// TwinCAT 3 PLC project PLC
// ProgramVersion: 3.1.4024.0
// libraries:
//   Tc2_MC2, * (Beckhoff Automation GmbH)
//   Tc2_Standard, * (Beckhoff Automation GmbH)
//   Tc2_System, * (Beckhoff Automation GmbH)
//   Tc2_Utilities, * (Beckhoff Automation GmbH)
//   Tc3_EventLogger, * (Beckhoff Automation GmbH)
//   Tc3_Module, * (Beckhoff Automation GmbH)
//   Util, * (System)
// project tree:
//   DUTs/ E_State.TcDUT, ST_CarrierSetpoint.TcDUT, ST_LEDButton.TcDUT, ST_MachineModuleInputs.TcDUT
//   / PlcTask.TcTTO (not stored)
//   POUs/ FB_CarrierStop.TcPOU, FB_CarrierReset.TcPOU, FB_CarrierAbsMove.TcPOU, FB_Machine.TcPOU, FB_Alarm.TcPOU, F_E_State_To_String.TcPOU, MAIN.TcPOU, PRG_LoadTwinSAFE.TcPOU
// real-time tasks:
//   TASK PlcTask: cycle T#10ms, priority 20, ADS port 350
// motion (NC):
//   TASK NC-Task 1 SAF: cycle T#2ms, priority 4, ADS port 501
//   TASK NC-Task 1 SVB: cycle T#10ms, priority 8, ADS port 511
//   AXIS X (id 1)
//     Dynamic: AccelerationMaximum=100000, DecelerationMaximum=100000, Acceleration=3082.5, Deceleration=3082.5, Jerk=9247.5
//     Velo: RefSearch=20.55, RefSync=20.55, SlowManual=102.75, FastManual=616.5, Fast=2055, Maximum=2055
//     OtherSettings: AllowMotionCmdToSlave=true
//     encoder EncType=19
//       EncPara: ScaleFactorNumerator=100, ScaleFactorDenominator=1048576, MaxCount=#xffffffff
//         SoftEndMinControl: Enable=true
//         SoftEndMaxControl: Enable=true, Range=2000
//     encoder EncId=129, EncType=5
//       EncPara: ScaleFactorNumerator=10, ScaleFactorDenominator=4096, Offset=-1035.7471, MaxCount=#xffffffff, ReferenceSystem=1
//         Inc: RefSoftSyncMask=#x0000ffff
//     drive DrvType=16
//       DrvPara: MaxCount=#xffffffff, DriveControlDWord=#x00020100
//         Analog: VeloReferenz=2260.5, VeloScale=32, TorqueSetpointScale=10, ScaleFactorActTorque=0.1
//         TimeComp: TaskDelayCycles=1
//     controller CtrType=1
//       CtrPara: PriorControlFactor=1
//         Observer: BandWidth=20
//   AXIS Z (id 2)
//     Dynamic: AccelerationMaximum=100000, DecelerationMaximum=100000, Acceleration=3082.5, Deceleration=3082.5, Jerk=9247.5
//     Velo: RefSearch=20.55, RefSync=20.55, SlowManual=102.75, FastManual=616.5, Fast=2055, Maximum=2055
//     OtherSettings: AllowMotionCmdToSlave=true
//     encoder EncType=19
//       EncPara: ScaleFactorNumerator=100, ScaleFactorDenominator=1048576, MaxCount=#xffffffff
//         SoftEndMinControl: Enable=true
//         SoftEndMaxControl: Enable=true, Range=1500
//     drive DrvType=16
//       DrvPara: MaxCount=#xffffffff, DriveControlDWord=#x00020100
//         Analog: VeloReferenz=2260.5, VeloScale=32, TorqueSetpointScale=10, ScaleFactorActTorque=0.1
//         TimeComp: TaskDelayCycles=1
//     controller CtrType=1
//       CtrPara: PriorControlFactor=1
//         Observer: BandWidth=20
// I/O:
//   DEVICE Real IO, AmsNetId 0.0.0.0.2.1
//     Term 1 (EK1200) [EK1200-5000 EtherCAT Power supply (2A E-Bus)]
//       Machine Safety Controller (EL6910) [EL6910, TwinSAFE PLC]
//       Operator Panel Safe In (EL1904) [EL1904, 4 Ch. Safety Input 24V, TwinSAFE]
//         modules: Module 1 (FSOES)
//   DEVICE Sim IO, AmsNetId 0.0.0.0.3.1
//     Machine A (EK1100) [EK1100 EtherCAT Coupler (2A E-Bus)]
//       Machine A Safe In (EL1904) [EL1904, 4 Ch. Safety Input 24V, TwinSAFE]
//         modules: Module 1 (FSOES)
//       Machine A Safe out (EL2904) [EL2904, 4 Ch. Safety Output 24V, 0.5A, TwinSAFE]
//         modules: Module 1 (FSOES), Module 2 (DO)
//       Robot (EL2002) [EL2002 2Ch. Dig. Output 24V, 0.5A]
//       Part Status (EL1002) [EL1002 2Ch. Dig. Input 24V, 3ms]
//     Machine B (EK1100) [EK1100 EtherCAT Coupler (2A E-Bus)]
//       Machine B Safe In (EL1904) [EL1904, 4 Ch. Safety Input 24V, TwinSAFE]
//         modules: Module 1 (FSOES)
//       Machine B Safe out (EL2904) [EL2904, 4 Ch. Safety Output 24V, 0.5A, TwinSAFE]
//         modules: Module 1 (FSOES), Module 2 (DO)
//       QC Check (EL3001) [EL3001 1Ch. Ana. Input +/-10V]
//     Machine C (EK1100) [EK1100 EtherCAT Coupler (2A E-Bus)]
//       Machine C Safe In (EL1904) [EL1904, 4 Ch. Safety Input 24V, TwinSAFE]
//         modules: Module 1 (FSOES)
//       Machine C Safe out (EL2904) [EL2904, 4 Ch. Safety Output 24V, 0.5A, TwinSAFE]
//         modules: Module 1 (FSOES), Module 2 (DO)
//       Bending (EL4001) [EL4001 1Ch. Ana. Output 0-10V, 12bit]
//     Machine D (EK1100) [EK1100 EtherCAT Coupler (2A E-Bus)]
//       Machine D Safe In (EL1904) [EL1904, 4 Ch. Safety Input 24V, TwinSAFE]
//         modules: Module 1 (FSOES)
//       Machine D Safe out (EL2904) [EL2904, 4 Ch. Safety Output 24V, 0.5A, TwinSAFE]
//         modules: Module 1 (FSOES), Module 2 (DO)
//       Carrier X Safety Encoder (EL5001-0090) [EL5001-0090 1Ch. SSI Encoder, TwinSAFE SC]
//         modules: Module 1 (EL5001-0090)
//       Carrier X Axis (EL7211-9014) [EL7211-9014 1Ch. MDP742 Servo motor output stage with OCT (50V, 4.5A RMS) and STO input]
//       Carrier Z Axis (EL7211-9014) [EL7211-9014 1Ch. MDP742 Servo motor output stage with OCT (50V, 4.5A RMS) and STO input]
//       Carrier Gripper (EL2002) [EL2002 2Ch. Dig. Output 24V, 0.5A]
//   DEVICE CP Buttons
// variable links:
//   Real IO <-> Sim IO/Machine A (EK1100)/Machine A Safe In (EL1904)
//     Term 1 (EK1200)/Machine Safety Controller (EL6910)/ConnectionInputs/TwinSafeGroup1.Machine A Safe In (EL1904) - Module 1 (FSOES)_32 TxPDO <-> Module 1 (FSOES)/RxPDO/FSOE
//     Term 1 (EK1200)/Machine Safety Controller (EL6910)/ConnectionOutputs/TwinSafeGroup1.Machine A Safe In (EL1904) - Module 1 (FSOES)_32 RxPDO <-> Module 1 (FSOES)/TxPDO/FSOE
//   Real IO <-> Sim IO/Machine B (EK1100)/Machine B Safe In (EL1904)
//     Term 1 (EK1200)/Machine Safety Controller (EL6910)/ConnectionOutputs/TwinSafeGroup1.Machine B Safe In (EL1904) - Module 1 (FSOES)_34 RxPDO <-> Module 1 (FSOES)/TxPDO/FSOE
//   Real IO <-> Sim IO/Machine B (EK1100)/Machine B Safe out (EL2904)
//     Term 1 (EK1200)/Machine Safety Controller (EL6910)/ConnectionInputs/TwinSafeGroup1.Machine B Safe out (EL2904) - Module 1 (FSOES)_35 TxPDO <-> Module 1 (FSOES)/RxPDO/FSOE
//   Real IO <-> Sim IO/Machine C (EK1100)/Machine C Safe In (EL1904)
//     Term 1 (EK1200)/Machine Safety Controller (EL6910)/ConnectionInputs/TwinSafeGroup1.Machine C Safe In (EL1904) - Module 1 (FSOES)_36 TxPDO <-> Module 1 (FSOES)/RxPDO/FSOE
//     Term 1 (EK1200)/Machine Safety Controller (EL6910)/ConnectionOutputs/TwinSafeGroup1.Machine C Safe In (EL1904) - Module 1 (FSOES)_36 RxPDO <-> Module 1 (FSOES)/TxPDO/FSOE
//   Real IO <-> Sim IO/Machine C (EK1100)/Machine C Safe out (EL2904)
//     Term 1 (EK1200)/Machine Safety Controller (EL6910)/ConnectionInputs/TwinSafeGroup1.Machine C Safe out (EL2904) - Module 1 (FSOES)_37 TxPDO <-> Module 1 (FSOES)/RxPDO/FSOE
//     Term 1 (EK1200)/Machine Safety Controller (EL6910)/ConnectionOutputs/TwinSafeGroup1.Machine C Safe out (EL2904) - Module 1 (FSOES)_37 RxPDO <-> Module 1 (FSOES)/TxPDO/FSOE
//   Real IO <-> Sim IO/Machine D (EK1100)/Carrier X Safety Encoder (EL5001-0090)
//     Term 1 (EK1200)/Machine Safety Controller (EL6910)/ConnectionInputs/TwinSafeGroup1.Carrier X Safety Encoder (EL5001-0090) - Module 1 (EL5001-0090)_48 TxPDO <-> Module 1 (EL5001-0090)/TSC Master Message/TSC
//     Term 1 (EK1200)/Machine Safety Controller (EL6910)/ConnectionOutputs/TwinSafeGroup1.Carrier X Safety Encoder (EL5001-0090) - Module 1 (EL5001-0090)_48 RxPDO <-> Module 1 (EL5001-0090)/TSC Slave Message/TSC
//   Sim IO <-> Real IO/Term 1 (EK1200)/Machine Safety Controller (EL6910)
//     Machine A (EK1100)/Machine A Safe out (EL2904)/Module 1 (FSOES)/RxPDO/FSOE <-> ConnectionInputs/TwinSafeGroup1.Machine A Safe out (EL2904) - Module 1 (FSOES)_33 TxPDO
//     Machine A (EK1100)/Machine A Safe out (EL2904)/Module 1 (FSOES)/TxPDO/FSOE <-> ConnectionOutputs/TwinSafeGroup1.Machine A Safe out (EL2904) - Module 1 (FSOES)_33 RxPDO
//     Machine B (EK1100)/Machine B Safe In (EL1904)/Module 1 (FSOES)/RxPDO/FSOE <-> ConnectionInputs/TwinSafeGroup1.Machine B Safe In (EL1904) - Module 1 (FSOES)_34 TxPDO
//     Machine B (EK1100)/Machine B Safe out (EL2904)/Module 1 (FSOES)/TxPDO/FSOE <-> ConnectionOutputs/TwinSafeGroup1.Machine B Safe out (EL2904) - Module 1 (FSOES)_35 RxPDO
//     Machine D (EK1100)/Machine D Safe In (EL1904)/Module 1 (FSOES)/RxPDO/FSOE <-> ConnectionInputs/TwinSafeGroup1.Machine D Safe In (EL1904) - Module 1 (FSOES)_38 TxPDO
//     Machine D (EK1100)/Machine D Safe In (EL1904)/Module 1 (FSOES)/TxPDO/FSOE <-> ConnectionOutputs/TwinSafeGroup1.Machine D Safe In (EL1904) - Module 1 (FSOES)_38 RxPDO
//     Machine D (EK1100)/Machine D Safe out (EL2904)/Module 1 (FSOES)/RxPDO/FSOE <-> ConnectionInputs/TwinSafeGroup1.Machine D Safe out (EL2904) - Module 1 (FSOES)_39 TxPDO
//     Machine D (EK1100)/Machine D Safe out (EL2904)/Module 1 (FSOES)/TxPDO/FSOE <-> ConnectionOutputs/TwinSafeGroup1.Machine D Safe out (EL2904) - Module 1 (FSOES)_39 RxPDO
//   (this object) <-> Sim IO/Machine D (EK1100)/Carrier X Axis (EL7211-9014)
//     Drive/Inputs/In/nDataIn1 <-> DRV Following error actual value/Following error actual value
//     Drive/Inputs/In/nDataIn3[0] <-> DRV Torque actual value/Torque actual value
//     Drive/Inputs/In/nDcOutputTime <-> InfoData/DcOutputShift
//     Drive/Inputs/In/nState1 <-> DRV Statusword/Statusword
//     Drive/Inputs/In/nState2 <-> DRV Statusword/Statusword @bit 8
//     Drive/Inputs/In/nState4 @bit 1 <-> WcState/InputToggle
//     Drive/Inputs/In/nState4 <-> WcState/WcState
//     Drive/Outputs/Out/nCtrl1 <-> DRV Controlword/Controlword
//     Drive/Outputs/Out/nCtrl2 <-> DRV Controlword/Controlword @bit 8
//     Drive/Outputs/Out/nDataOut1 <-> DRV Target position/Target position
//     EL7211/Inputs/In/nDataIn1 <-> FB Position/Position
//     EL7211/Inputs/In/nDcInputTime <-> InfoData/DcInputShift
//     EL7211/Inputs/In/nState4 @bit 1 <-> WcState/InputToggle
//     EL7211/Inputs/In/nState4 <-> WcState/WcState
//   (this object) <-> Sim IO/Machine D (EK1100)/Carrier X Safety Encoder (EL5001-0090)
//     EL5001-0090/Inputs/In/nDataIn1 <-> SSI Inputs/Counter value
//     EL5001-0090/Inputs/In/nState1 <-> SSI Inputs/Status/Data error
//     EL5001-0090/Inputs/In/nState1 @bit 1 <-> SSI Inputs/Status/Frame error
//     EL5001-0090/Inputs/In/nState1 @bit 2 <-> SSI Inputs/Status/Power failure
//     EL5001-0090/Inputs/In/nState2 @bit 5 <-> SSI Inputs/Status/Sync error
//     EL5001-0090/Inputs/In/nState2 @bit 6 <-> SSI Inputs/Status/TxPDO State
//     EL5001-0090/Inputs/In/nState2 @bit 7 <-> SSI Inputs/Status/TxPDO Toggle
//     EL5001-0090/Inputs/In/nState4 @bit 1 <-> WcState/InputToggle
//     EL5001-0090/Inputs/In/nState4 <-> WcState/WcState
//   (this object) <-> Sim IO/Machine D (EK1100)/Carrier Z Axis (EL7211-9014)
//     Drive/Inputs/In/nDataIn1 <-> DRV Following error actual value/Following error actual value
//     Drive/Inputs/In/nDataIn3[0] <-> DRV Torque actual value/Torque actual value
//     Drive/Inputs/In/nDcOutputTime <-> InfoData/DcOutputShift
//     Drive/Inputs/In/nState1 <-> DRV Statusword/Statusword
//     Drive/Inputs/In/nState2 <-> DRV Statusword/Statusword @bit 8
//     Drive/Inputs/In/nState4 @bit 1 <-> WcState/InputToggle
//     Drive/Inputs/In/nState4 <-> WcState/WcState
//     Drive/Outputs/Out/nCtrl1 <-> DRV Controlword/Controlword
//     Drive/Outputs/Out/nCtrl2 <-> DRV Controlword/Controlword @bit 8
//     Drive/Outputs/Out/nDataOut1 <-> DRV Target position/Target position
//     EL7211/Inputs/In/nDataIn1 <-> FB Position/Position
//     EL7211/Inputs/In/nDcInputTime <-> InfoData/DcInputShift
//     EL7211/Inputs/In/nState4 @bit 1 <-> WcState/InputToggle
//     EL7211/Inputs/In/nState4 <-> WcState/WcState
//   (this object) <-> Real IO
//     Term 1 (EK1200)/Machine Safety Controller (EL6910)/ConnectionInputs/TwinSafeGroup1.Operator Panel Safe In (EL1904) - Module 1 (FSOES)_43 TxPDO <-> Term 1 (EK1200)/Operator Panel Safe In (EL1904)/Module 1 (FSOES)/RxPDO/FSOE
//     Term 1 (EK1200)/Machine Safety Controller (EL6910)/ConnectionOutputs/TwinSafeGroup1.Operator Panel Safe In (EL1904) - Module 1 (FSOES)_43 RxPDO <-> Term 1 (EK1200)/Operator Panel Safe In (EL1904)/Module 1 (FSOES)/TxPDO/FSOE
//     Term 1 (EK1200)/Operator Panel Safe In (EL1904)/Module 1 (FSOES)/RxPDO/FSOE <-> Term 1 (EK1200)/Machine Safety Controller (EL6910)/ConnectionInputs/TwinSafeGroup1.Operator Panel Safe In (EL1904) - Module 1 (FSOES)_43 TxPDO
//     Term 1 (EK1200)/Operator Panel Safe In (EL1904)/Module 1 (FSOES)/TxPDO/FSOE <-> Term 1 (EK1200)/Machine Safety Controller (EL6910)/ConnectionOutputs/TwinSafeGroup1.Operator Panel Safe In (EL1904) - Module 1 (FSOES)_43 RxPDO
//   PLC Instance <-> CP Buttons/Box 0 (CPX8XX)
//     PlcTask Inputs/MAIN.Machine.LocalEstop <-> Term 1 (CPx9xx-4)/Channel 1/Estop
//     PlcTask Inputs/MAIN.Machine.Reset.Button <-> Term 1 (CPx9xx-4)/Channel 1/BlueBtn
//     PlcTask Inputs/MAIN.Machine.Start.Button <-> Term 1 (CPx9xx-4)/Channel 1/GreenBtn
//     PlcTask Inputs/MAIN.Machine.Stop.Button <-> Term 1 (CPx9xx-4)/Channel 1/RedBtn
//     PlcTask Outputs/MAIN.Machine.Reset.LED <-> Term 1 (CPx9xx-4)/Channel 1/BlueBtnLight
//     PlcTask Outputs/MAIN.Machine.Start.LED <-> Term 1 (CPx9xx-4)/Channel 1/GreenBtnLight
//     PlcTask Outputs/MAIN.Machine.Stop.LED <-> Term 1 (CPx9xx-4)/Channel 1/RedBtnLight
//   PLC Instance <-> Real IO/Term 1 (EK1200)/Machine Safety Controller (EL6910)
//     PlcTask Inputs/MAIN.Machine.TwinSAFEGroupState <-> TwinSAFE Group Info Data/TwinSafeGroup1 Info Data/State
//     PlcTask Inputs/MAIN.Machine.TwinSAFE_Machine_A_Estop_State <-> Function Block Info Data/TwinSafeGroup1.MachineA.Machine_A.FBEstop1 Info Data/State
//     PlcTask Inputs/MAIN.Machine.TwinSAFE_Machine_B_Estop_State <-> Function Block Info Data/TwinSafeGroup1.MachineB.Machine_B.FBEstop1 Info Data/State
//     PlcTask Inputs/MAIN.Machine.TwinSAFE_Machine_C_Estop_State <-> Function Block Info Data/TwinSafeGroup1.MachineC.Machine_C.FBEstop1 Info Data/State
//     PlcTask Inputs/MAIN.Machine.TwinSAFE_Machine_D_Estop_State <-> Function Block Info Data/TwinSafeGroup1.MachineD.Machine_D_Estop Info Data/State
//     PlcTask Inputs/PRG_LoadTwinSAFE.ProjectCRC <-> Device Info Data/Project CRC
//     PlcTask Inputs/PRG_LoadTwinSAFE.WcState <-> WcState/WcState
//     PlcTask Outputs/MAIN.Machine.TwinSAFEGroupErrAck <-> StandardOutputs/TwinSafeGroup1.ErrorAcknowledgement_1
//     PlcTask Outputs/MAIN.Machine.TwinSAFEGroupRun <-> StandardOutputs/TwinSafeGroup1.Run_2
//     PlcTask Outputs/MAIN.Machine.TwinSAFE_ResetAllEstopZones <-> StandardOutputs/TwinSafeGroup1.ResetAllZones_55
//     PlcTask Outputs/MAIN.Machine.TwinSAFE_X_Axis_ActPos <-> StandardOutputs/TwinSafeGroup1.X_ActPosFromPLC_51
//   PLC Instance <-> Sim IO/Machine A (EK1100)/Machine A Safe In (EL1904)
//     PlcTask Inputs/MAIN.Machine.MachineAIn.EstopBtn <-> Module 1 (FSOES)/TxPDO/FSOE/E-Stop PB
//     PlcTask Inputs/MAIN.Machine.MachineAIn.LightCurtain <-> Module 1 (FSOES)/TxPDO/FSOE/Light Curtain
//   PLC Instance <-> Sim IO/Machine B (EK1100)/Machine B Safe In (EL1904)
//     PlcTask Inputs/MAIN.Machine.MachineBIn.EstopBtn <-> Module 1 (FSOES)/TxPDO/FSOE/E-Stop PB
//     PlcTask Inputs/MAIN.Machine.MachineBIn.LightCurtain <-> Module 1 (FSOES)/TxPDO/FSOE/Light Curtain
//   PLC Instance <-> Sim IO/Machine C (EK1100)/Machine C Safe In (EL1904)
//     PlcTask Inputs/MAIN.Machine.MachineCIn.EstopBtn <-> Module 1 (FSOES)/TxPDO/FSOE/E-Stop PB
//     PlcTask Inputs/MAIN.Machine.MachineCIn.LightCurtain <-> Module 1 (FSOES)/TxPDO/FSOE/Light Curtain
//   PLC Instance <-> Sim IO/Machine D (EK1100)/Carrier Gripper (EL2002)
//     PlcTask Outputs/MAIN.Machine.Machine_D_Carrier_Gripper <-> Fingers/Output
//   PLC Instance <-> Sim IO/Machine D (EK1100)/Machine D Safe In (EL1904)
//     PlcTask Inputs/MAIN.Machine.MachineDIn.EstopBtn <-> Module 1 (FSOES)/TxPDO/FSOE/E-Stop PB
//   PLC Instance <-> NC-Task 1 SAF/Axes/X
//     PlcTask Inputs/MAIN.Machine.X_Axis.NcToPlc <-> Outputs/ToPlc
//     PlcTask Outputs/MAIN.Machine.X_Axis.PlcToNc <-> Inputs/FromPlc
//   PLC Instance <-> NC-Task 1 SAF/Axes/Z
//     PlcTask Inputs/MAIN.Machine.Z_Axis.NcToPlc <-> Outputs/ToPlc
//     PlcTask Outputs/MAIN.Machine.Z_Axis.PlcToNc <-> Inputs/FromPlc

// ---- DUTs/E_State.TcDUT
{attribute 'qualified_only'}
{attribute 'strict'}
TYPE
	E_State :
	(
		Init := 0,
		Idel,
		Enable,
		MoveToHome,			// Move X and Z to home poisition
		WaitForAToBeReady,	// Wait at home postion for A to be ready
		MoveToAPickPos,		// Move X and Z to A position
		PickFromA,			// Close Grippers
		MoveToBWaitPos,		// Move X and Z to safe B position
		WaitForBToBeReady,
		MoveToBPlacePosition,	// Move X and Z to B Position
		PlaceOnB,				// Open grippers
		MoveToBWorkPos,			// Move Carrier up and out of the way for B to do work
		BDoingWork,
		MoveToBPickPos,	// Move carrier to B to retreive part
		PickPartFromB,	// Close grippers
		MoveToCWaitPos,	// Move to C wait position
		WaitForCToBeReady,
		MoveToCPlacePos,	// Move down to C place position
		PlaceOnC,			// Open Grippers
		MoveToCWorkPos,		// Move Carrier up and out of the wayt for C to do work
		CDoingWork,
		Stopping,
		Stopped,
		Error,
		Reseting
	);
END_TYPE

// ---- DUTs/ST_CarrierSetpoint.TcDUT
TYPE
	ST_CarrierSetpoint :
	STRUCT
		X_Pos	: LREAL;
		X_Velo	: LREAL;
		Z_Pos	: LREAL;
		Z_Velo	: LREAL;
	END_STRUCT
END_TYPE

// ---- DUTs/ST_LEDButton.TcDUT
TYPE
	ST_LEDButton :
	STRUCT
		Button	AT %I*	: BOOL;
		LED		AT %Q*	: BOOL;
	END_STRUCT
END_TYPE

// ---- DUTs/ST_MachineModuleInputs.TcDUT
TYPE
	ST_MachineModuleInputs :
	STRUCT
		EstopBtn		AT %I*	: BOOL;
		LightCurtain	AT %I*	: BOOL;
	END_STRUCT
END_TYPE

// ---- POUs/FB_CarrierStop.TcPOU
FUNCTION_BLOCK FB_CarrierStop
VAR_INPUT
	Execute : BOOL;
END_VAR
VAR_OUTPUT
	Busy	: BOOL;
	Done	: BOOL;
	Error	: BOOL;
END_VAR
VAR
	_Decel : LREAL := 100000.0;

	X_AxisHalt	: MC_Halt;
	Z_AxisHalt	: MC_Halt;

	{attribute 'hide'}
	_X_Axis : POINTER TO AXIS_REF;
	{attribute 'hide'}
	_Z_Axis : POINTER TO AXIS_REF;

END_VAR

IF _X_Axis = 0 OR _Z_Axis = 0 THEN
	RETURN;
END_IF

X_AxisHalt(Axis			:= _X_Axis^,
			Deceleration := _Decel,
			Execute		:= Execute);

Z_AxisHalt(Axis			:= _Z_Axis^,
			Deceleration := _Decel,
			Execute		:= Execute);

Busy := X_AxisHalt.Busy OR Z_AxisHalt.Busy;

Done := X_AxisHalt.Done AND Z_AxisHalt.Done;

Error := X_AxisHalt.Error OR Z_AxisHalt.Error;

PROPERTY Decel : LREAL
GET
Decel := _Decel;
END_GET
SET
_Decel := Decel;
END_SET
END_PROPERTY

PROPERTY X_AxisRef : POINTER TO AXIS_REF
GET
X_AxisRef := _X_Axis;
END_GET
SET
_X_Axis := X_AxisRef;
END_SET
END_PROPERTY

PROPERTY Z_AxisRef : POINTER TO AXIS_REF
GET
Z_AxisRef := _Z_Axis;
END_GET
SET
_Z_Axis := Z_AxisRef;
END_SET
END_PROPERTY

END_FUNCTION_BLOCK

// ---- POUs/FB_CarrierReset.TcPOU
FUNCTION_BLOCK FB_CarrierReset
VAR_INPUT
	Execute : BOOL;
END_VAR
VAR_OUTPUT
	Busy	: BOOL;
	Done	: BOOL;
	Error	: BOOL;
END_VAR
VAR
	X_AxisReset	: MC_Reset;
	Z_AxisReset	: MC_Reset;

	{attribute 'hide'}
	_X_Axis : POINTER TO AXIS_REF;
	{attribute 'hide'}
	_Z_Axis		: POINTER TO AXIS_REF;
	_SetPoint	: ST_CarrierSetpoint;
END_VAR

IF _X_Axis = 0 OR _Z_Axis = 0 THEN
	RETURN;
END_IF

X_AxisReset(Axis	:= _X_Axis^,
			Execute := Execute AND _X_Axis^.Status.Error);

Z_AxisReset(Axis	:= _Z_Axis^,
			Execute := Execute AND _Z_Axis^.Status.Error);

Busy := X_AxisReset.Busy OR Z_AxisReset.Busy;

Done := X_AxisReset.Done AND Z_AxisReset.Done;

Error := X_AxisReset.Error OR Z_AxisReset.Error;

PROPERTY X_AxisRef : POINTER TO AXIS_REF
GET
X_AxisRef := _X_Axis;
END_GET
SET
_X_Axis := X_AxisRef;
END_SET
END_PROPERTY

PROPERTY Z_AxisRef : POINTER TO AXIS_REF
GET
Z_AxisRef := _Z_Axis;
END_GET
SET
_Z_Axis := Z_AxisRef;
END_SET
END_PROPERTY

END_FUNCTION_BLOCK

// ---- POUs/FB_CarrierAbsMove.TcPOU
FUNCTION_BLOCK FB_CarrierAbsMove
VAR_INPUT
	Execute : BOOL;
END_VAR
VAR_OUTPUT
	Busy	: BOOL;
	Done	: BOOL;
	Error	: BOOL;
END_VAR
VAR
	X_AxisMoveAbs	: MC_MoveAbsolute;
	Z_AxisMoveAbs	: MC_MoveAbsolute;

	{attribute 'hide'}
	_X_Axis : POINTER TO AXIS_REF;
	{attribute 'hide'}
	_Z_Axis : POINTER TO AXIS_REF;
	{attribute 'hide'}
	_SetPoint : ST_CarrierSetpoint;
END_VAR

IF _X_Axis = 0 OR _Z_Axis = 0 THEN
	RETURN;
END_IF

X_AxisMoveAbs(Axis		:= _X_Axis^,
				Execute := Execute,
				Position := _SetPoint.X_Pos,
				Velocity := _SetPoint.X_Velo);

Z_AxisMoveAbs(Axis		:= _Z_Axis^,
				Execute := Execute,
				Position := _SetPoint.Z_Pos,
				Velocity := _SetPoint.Z_Velo);

Busy := X_AxisMoveAbs.Busy OR Z_AxisMoveAbs.Busy;

Done := X_AxisMoveAbs.Done AND Z_AxisMoveAbs.Done;

Error := X_AxisMoveAbs.Error OR Z_AxisMoveAbs.Error OR X_AxisMoveAbs.CommandAborted OR Z_AxisMoveAbs.CommandAborted;

PROPERTY SetPoint : ST_CarrierSetpoint
GET
SetPoint := _SetPoint;
END_GET
SET
_SetPoint := SetPoint;
END_SET
END_PROPERTY

PROPERTY X_AxisRef : POINTER TO AXIS_REF
GET
X_AxisRef := _X_Axis;
END_GET
SET
_X_Axis := X_AxisRef;
END_SET
END_PROPERTY

PROPERTY Z_AxisRef : POINTER TO AXIS_REF
GET
Z_AxisRef := _Z_Axis;
END_GET
SET
_Z_Axis := Z_AxisRef;
END_SET
END_PROPERTY

END_FUNCTION_BLOCK

// ---- POUs/FB_Machine.TcPOU
FUNCTION_BLOCK FB_Machine
VAR_INPUT
END_VAR
VAR_OUTPUT
END_VAR
VAR
	//Alarms
	AlarmLocalEstopBtn	: FB_Alarm;
	AlarmAEstopBtn		: FB_Alarm;
	AlarmBEstopBtn		: FB_Alarm;
	AlarmCEstopBtn		: FB_Alarm;
	AlarmDEstopBtn		: FB_Alarm;

	AlarmALightCurtain	: FB_Alarm;
	AlarmBLightCurtain	: FB_Alarm;
	AlarmCLightCurtain	: FB_Alarm;

	AlarmXNotReady	: FB_Alarm;
	AlarmZNotReady	: FB_Alarm;

	AlarmXAxisError	: FB_Alarm;
	AlarmZAxisError	: FB_Alarm;
	
	AlarmAEstopTripped	:FB_Alarm;
	AlarmBEstopTripped	:FB_Alarm;
	AlarmCEstopTripped	:FB_Alarm;
	AlarmDEstopTripped	:FB_Alarm;

	//Buttons
	Start		: ST_LEDButton;
	HMI_Start	: ST_LEDButton;
	rtStart		: R_TRIG;
	Stop		: ST_LEDButton;
	HMI_Stop	: ST_LEDButton;
	rtStop		: R_TRIG;
	Reset		: ST_LEDButton;
	HMI_Reset	: ST_LEDButton;
	rtReset		: R_TRIG;

	//Inputs
	LocalEstop AT %I*	: BOOL;
	MachineAIn			: ST_MachineModuleInputs;
	MachineBIn			: ST_MachineModuleInputs;
	MachineCIn			: ST_MachineModuleInputs;
	MachineDIn			: ST_MachineModuleInputs;

	//Overide
	Override : LREAL := 50.0;

	TwinSAFEGroupRun			AT %Q*	: BOOL := TRUE;
	TwinSAFEGroupErrAck			AT %Q*	: BOOL;
	TwinSAFEGroupState			AT %I*	: USINT;
	TwinSAFE_X_Axis_ActPos		AT %Q*	: UDINT;
	TwinSAFE_ResetAllEstopZones	AT %Q*	: BOOL;

	TwinSAFE_Machine_A_Estop_State	AT %I*	: USINT;
	TwinSAFE_Machine_B_Estop_State	AT %I*	: USINT;
	TwinSAFE_Machine_C_Estop_State	AT %I*	: USINT;
	TwinSAFE_Machine_D_Estop_State	AT %I*	: USINT;

	AxisInError : BOOL; //One or more axis in error

	X_Axis			: AXIS_REF;
	Z_Axis			: AXIS_REF;
	fbCarrierReset	: FB_CarrierReset;

	fbCarrierStop : FB_CarrierStop;

	StateToReturnToAfterStop	: E_State;
	lastState					: E_State;
	previousState				: E_State;
	State						: E_State;
	NextState					: E_State;

	//HMI Display               		
	sPreviouseState : STRING;

	sState : STRING;

	sNextState : STRING;

	fbMoveCarrier		: FB_CarrierAbsMove;
	HomePosSetPoint		: ST_CarrierSetPoint	:= (X_Pos := 100, X_Velo := 500, Z_Pos := 100, Z_Velo := 800);
	APickPosSetPoint	: ST_CarrierSetPoint	:= (X_Pos := 290, X_Velo := 500, Z_Pos := 1100, Z_Velo := 800);
	BWaitPosSetpoint	: ST_CarrierSetPoint	:= (X_Pos := 600, X_Velo := 500, Z_Pos := 100, Z_Velo := 800);
	BPlacePosSetPoint	: ST_CarrierSetPoint	:= (X_Pos := 1000, X_Velo := 500, Z_Pos := 1200, Z_Velo := 800);
	BWorkPosSetPoint	: ST_CarrierSetPoint	:= (X_Pos := 1000, X_Velo := 500, Z_Pos := 100, Z_Velo := 800);
	BPickPosSetPoint	: ST_CarrierSetPoint	:= (X_Pos := 1000, X_Velo := 500, Z_Pos := 1200, Z_Velo := 800);
	CWaitPosSetPoint	: ST_CarrierSetPoint	:= (X_Pos := 1350, X_Velo := 500, Z_Pos := 100, Z_Velo := 800);
	CPlacePosSetPoint	: ST_CarrierSetPoint	:= (X_Pos := 1700, X_Velo := 500, Z_Pos := 1000, Z_Velo := 800);
	CWorkPosSetPoint	: ST_CarrierSetPoint	:= (X_Pos := 1800, X_Velo := 500, Z_Pos := 100, Z_Velo := 800);

	//Machine A                 		
	WaitTimeForAToBeReady : TIME := T#1S;

	//Machine B             		
	WaitTimeForBtoBeReady	: TIME	:= T#1.5S;
	BDoingWorkTime			: TIME	:= T#2S;

	//Machine C             			
	WaitTimeForCtoBeReady	: TIME	:= T#0.5S;
	CDoingWorkTime			: TIME	:= T#750MS;

	//Machine D
	Machine_D_Carrier_Gripper AT %Q* : BIT;

	iResetingStep : UDINT;

END_VAR

IF NOT M_Init() THEN
	RETURN;
END_IF

rtStart(CLK := Start.Button OR HMI_Start.Button);
rtStop(CLK := Stop.Button OR HMI_Stop.Button);
rtReset(CLK := Reset.Button OR HMI_Reset.Button);

M_HMI_Display();

CASE State OF
	E_State.Init:
		fbMoveCarrier.X_AxisRef	:= ADR(X_Axis);
		fbMoveCarrier.Z_AxisRef	:= ADR(Z_Axis);
		fbMoveCarrier(Execute := FALSE);
		Machine_D_Carrier_Gripper := FALSE;

		fbCarrierReset(Execute := FALSE);
		fbCarrierReset.X_AxisRef	:= ADR(X_Axis);
		fbCarrierReset.Z_AxisRef	:= ADR(Z_Axis);

		fbCarrierStop(Execute := FALSE);
		fbCarrierStop.X_AxisRef	:= ADR(X_Axis);
		fbCarrierStop.Z_AxisRef	:= ADR(Z_Axis);

		State			:= E_State.Idel;
		NextState		:= E_State.Idel;
		iResetingStep	:= 0;
	E_State.Idel:
		NextState := E_State.Enable;

		IF TwinSAFEGroupState = 1 AND NOT AxisInError THEN
			IF rtStart.Q THEN
				State := E_State.Enable;
			ELSIF rtReset.Q THEN
				State := E_State.Reseting;
			ELSIF AxisInError THEN
				State := E_State.Error;
			END_IF
		ELSE
			State := E_State.Error;
		END_IF

	E_State.Enable:
		NextState := E_State.MoveToHome;

		IF TwinSAFEGroupState = 1 THEN
			State := E_State.MoveToHome;
		ELSIF AxisInError OR TwinSAFEGroupState <> 1 THEN
			State := E_State.Error;
		END_IF

	E_State.MoveToHome:
		NextState					:= E_State.WaitForAToBeReady;
		StateToReturnToAfterStop	:= State;
		fbMoveCarrier.SetPoint		:= HomePosSetPoint;
		fbMoveCarrier(Execute := TRUE);

		IF fbMoveCarrier.Done THEN
			fbMoveCarrier(Execute := FALSE);
			State := E_State.WaitForAToBeReady;
		ELSIF fbMoveCarrier.Error THEN
			State := E_State.Error;
		END_IF

	E_State.WaitForAToBeReady:
		NextState					:= E_State.MoveToAPickPos;
		StateToReturnToAfterStop	:= State;

		IF M_ProcessDelay(WaitTimeForAToBeReady) THEN
			State := E_State.MoveToAPickPos;
		END_IF

	E_State.MoveToAPickPos:
		NextState					:= E_State.PickFromA;
		StateToReturnToAfterStop	:= State;
		fbMoveCarrier.SetPoint		:= APickPosSetPoint;
		fbMoveCarrier(Execute := TRUE);

		IF fbMoveCarrier.Done THEN
			fbMoveCarrier(Execute := FALSE);
			State := E_State.PickFromA;
		ELSIF fbMoveCarrier.Error THEN
			State := E_State.Error;
		END_IF

	E_State.PickFromA:
		NextState					:= E_State.MoveToBWaitPos;
		StateToReturnToAfterStop	:= State;

		IF M_CloseGripper() THEN
			State := E_State.MoveToBWaitPos;
		END_IF

	E_State.MoveToBWaitPos:
		NextState					:= E_State.WaitForBToBeReady;
		StateToReturnToAfterStop	:= State;
		fbMoveCarrier.SetPoint		:= BWaitPosSetpoint;
		fbMoveCarrier(Execute := TRUE);

		IF fbMoveCarrier.Done THEN
			fbMoveCarrier(Execute := FALSE);
			State := E_State.WaitForBToBeReady;
		ELSIF fbMoveCarrier.Error THEN
			State := E_State.Error;
		END_IF

	E_State.WaitForBToBeReady:
		NextState					:= E_State.MoveToBPlacePosition;
		StateToReturnToAfterStop	:= State;

		IF M_ProcessDelay(WaitTimeForBtoBeReady) THEN
			State := E_State.MoveToBPlacePosition;
		END_IF

	E_State.MoveToBPlacePosition:
		NextState					:= E_State.PlaceOnB;
		StateToReturnToAfterStop	:= State;
		fbMoveCarrier.SetPoint		:= BPlacePosSetPoint;
		fbMoveCarrier(Execute := TRUE);

		IF fbMoveCarrier.Done THEN
			fbMoveCarrier(Execute := FALSE);
			State := E_State.PlaceOnB;
		ELSIF fbMoveCarrier.Error THEN
			State := E_State.Error;
		END_IF

	E_State.PlaceOnB:
		NextState					:= E_State.MoveToBWorkPos;
		StateToReturnToAfterStop	:= State;

		IF M_OpenGripper() THEN
			State := E_State.MoveToBWorkPos;
		END_IF

	E_State.MoveToBWorkPos:
		NextState					:= E_State.BDoingWork;
		StateToReturnToAfterStop	:= State;
		fbMoveCarrier.SetPoint		:= BWorkPosSetPoint;
		fbMoveCarrier(Execute := TRUE);

		IF fbMoveCarrier.Done THEN
			fbMoveCarrier(Execute := FALSE);
			State := E_State.BDoingWork;
		ELSIF fbMoveCarrier.Error THEN
			State := E_State.Error;
		END_IF

	E_State.BDoingWork:
		NextState					:= E_State.MoveToBPickPos;
		StateToReturnToAfterStop	:= State;

		IF M_ProcessDelay(BDoingWorkTime) THEN
			State := E_State.MoveToBPickPos;
		END_IF

	E_State.MoveToBPickPos:
		NextState					:= E_State.PickPartFromB;
		StateToReturnToAfterStop	:= State;
		fbMoveCarrier.SetPoint		:= BPickPosSetPoint;
		fbMoveCarrier(Execute := TRUE);

		IF fbMoveCarrier.Done THEN
			fbMoveCarrier(Execute := FALSE);
			State := E_State.PickPartFromB;
		ELSIF fbMoveCarrier.Error THEN
			State := E_State.Error;
		END_IF

	E_State.PickPartFromB:
		NextState					:= E_State.MoveToCWaitPos;
		StateToReturnToAfterStop	:= State;

		IF M_CloseGripper() THEN
			State := E_State.MoveToCWaitPos;
		END_IF

	E_State.MoveToCWaitPos:
		NextState					:= E_State.WaitForCToBeReady;
		StateToReturnToAfterStop	:= State;
		fbMoveCarrier.SetPoint		:= CWaitPosSetPoint;
		fbMoveCarrier(Execute := TRUE);

		IF fbMoveCarrier.Done THEN
			fbMoveCarrier(Execute := FALSE);
			State := E_State.WaitForCToBeReady;
		ELSIF fbMoveCarrier.Error THEN
			State := E_State.Error;
		END_IF

	E_State.WaitForCToBeReady:
		NextState					:= E_State.MoveToCPlacePos;
		StateToReturnToAfterStop	:= State;

		IF M_ProcessDelay(WaitTimeForCtoBeReady) THEN
			State := E_State.MoveToCPlacePos;
		END_IF

	E_State.MoveToCPlacePos:
		NextState					:= E_State.PlaceOnC;
		StateToReturnToAfterStop	:= State;
		fbMoveCarrier.SetPoint		:= CPlacePosSetPoint;
		fbMoveCarrier(Execute := TRUE);

		IF fbMoveCarrier.Done THEN
			fbMoveCarrier(Execute := FALSE);
			State := E_State.PlaceOnC;
		ELSIF fbMoveCarrier.Error THEN
			State := E_State.Error;
		END_IF

	E_State.PlaceOnC:
		NextState					:= E_State.MoveToCWorkPos;
		StateToReturnToAfterStop	:= State;

		IF M_OpenGripper() THEN
			State := E_State.MoveToCWorkPos;
		END_IF

	E_State.MoveToCWorkPos:
		NextState					:= E_State.CDoingWork;
		StateToReturnToAfterStop	:= State;
		fbMoveCarrier.SetPoint		:= CWorkPosSetPoint;
		fbMoveCarrier(Execute := TRUE);

		IF fbMoveCarrier.Done THEN
			fbMoveCarrier(Execute := FALSE);
			State := E_State.CDoingWork;
		ELSIF fbMoveCarrier.Error THEN
			State := E_State.Error;
		END_IF

	E_State.CDoingWork:
		NextState					:= E_State.MoveToHome;
		StateToReturnToAfterStop	:= State;

		IF M_ProcessDelay(CDoingWorkTime) THEN
			State := E_State.MoveToHome;
		END_IF

	E_State.Stopping:
		NextState := E_State.Stopped;
		fbCarrierStop(Execute := TRUE);

		IF fbCarrierStop.Done THEN
			fbCarrierStop(Execute := FALSE);
			State := E_State.Stopped;
		ELSIF fbCarrierStop.Error THEN
			State := E_State.Error;
		END_IF

	E_State.Stopped:
		NextState := StateToReturnToAfterStop;

		IF rtStart.Q THEN
			fbMoveCarrier(Execute := FALSE);
			State := StateToReturnToAfterStop;
		END_IF

	E_State.Error:
		NextState := E_State.Reseting;

		IF rtReset.Q THEN
			State := E_State.Reseting;
		END_IF

	E_State.Reseting:
		NextState := E_State.Init;

		CASE iResetingStep OF
			0: //Toggle TS group Err ack
				TwinSAFEGroupErrAck	:= TRUE;
				iResetingStep		:= 10;

			10: //Clear axis error
				fbCarrierReset(Execute := TRUE);
				TwinSAFEGroupErrAck := FALSE;

				IF NOT fbCarrierReset.Busy THEN
					fbCarrierReset(Execute := FALSE);
					State := E_State.Init;
				END_IF
		END_CASE

END_CASE

M_AxisPower();
M_BtnLights();
M_ToTwinSAFE();
M_Alarms();

METHOD M_Alarms
AlarmLocalEstopBtn(AlarmState := LocalEstop);
AlarmAEstopBtn(AlarmState := NOT MachineAIn.EstopBtn);
AlarmBEstopBtn(AlarmState := NOT MachineBIn.EstopBtn);
AlarmCEstopBtn(AlarmState := NOT MachineCIn.EstopBtn);
AlarmDEstopBtn(AlarmState := NOT MachineDIn.EstopBtn);

AlarmALightCurtain(AlarmState := NOT MachineAIn.LightCurtain);
AlarmBLightCurtain(AlarmState := NOT MachineBIn.LightCurtain);
AlarmCLightCurtain(AlarmState := NOT MachineCIn.LightCurtain);

X_Axis.ReadStatus();
Z_Axis.ReadStatus();

AlarmXNotReady(AlarmState := X_Axis.Status.ErrorID = 16#4650);
AlarmZNotReady(AlarmState := Z_Axis.Status.ErrorID = 16#4650);

AlarmXAxisError(AlarmState := X_Axis.Status.ErrorID <> 16#4650 AND X_Axis.Status.ErrorID <> 0);
AlarmZAxisError(AlarmState := Z_Axis.Status.ErrorID <> 16#4650 AND Z_Axis.Status.ErrorID <> 0);

AlarmAEstopTripped(AlarmState := TwinSAFE_Machine_A_Estop_State<>1);
AlarmBEstopTripped(AlarmState := TwinSAFE_Machine_B_Estop_State<>1);
AlarmCEstopTripped(AlarmState := TwinSAFE_Machine_C_Estop_State<>1);
AlarmDEstopTripped(AlarmState := TwinSAFE_Machine_D_Estop_State<>1);
END_METHOD

METHOD M_AxisPower : BOOL
VAR_INPUT
END_VAR
VAR_INST
	X_Power	: MC_Power;
	Z_Power	: MC_Power;
END_VAR
X_Power(Axis			:= X_Axis,
		Enable			:= TRUE,
		Enable_Positive := TRUE,
		Enable_Negative := TRUE,
		Override		:= Override);

Z_Power(Axis			:= Z_Axis,
		Enable			:= TRUE,
		Enable_Positive := TRUE,
		Enable_Negative := TRUE,
		Override		:= Override);

X_Axis.ReadStatus();
Z_Axis.ReadStatus();

AxisInError := X_Axis.Status.Error OR Z_Axis.Status.Error;
END_METHOD

METHOD M_BtnLights
VAR_INPUT
END_VAR
VAR_INST
	StartLEDBlink	: BLINK;
	ResetLEDBlink	: BLINK;
	StopLEDBlink	: BLINK;
END_VAR
//Buttons
//Start
CASE State OF
	E_State.Init:
		Start.LED := FALSE;
	E_State.Idel:
		StartLEDBlink.TIMEHIGH	:= T#1S;
		StartLEDBlink.TIMELOW	:= T#1S;
		Start.LED				:= StartLEDBlink.out;
	E_State.Enable:
		StartLEDBlink.TIMEHIGH	:= T#500MS;
		StartLEDBlink.TIMELOW	:= T#500MS;
		Start.LED				:= StartLEDBlink.out;
	E_State.MoveToHome..E_State.CDoingWork:
		Start.LED := TRUE;
	E_State.Stopping:
		Start.LED := FALSE;
	E_State.Stopped:
		StartLEDBlink.TIMEHIGH	:= T#200MS;
		StartLEDBlink.TIMELOW	:= T#200MS;
		Start.LED				:= StartLEDBlink.out;
	E_State.Error..E_State.Reseting:
		Start.LED := FALSE;
END_CASE

HMI_Start.LED := Start.LED;
StartLEDBlink(ENABLE := TRUE);

//Reset
CASE State OF
	E_State.Init..E_State.CDoingWork:
		Reset.LED := FALSE;
	E_State.Error:
		ResetLEDBlink.TIMEHIGH	:= T#1S;
		ResetLEDBlink.TIMELOW	:= T#1S;
		Reset.LED				:= ResetLEDBlink.OUT;
	E_State.Reseting:
		ResetLEDBlink.TIMEHIGH	:= T#500MS;
		ResetLEDBlink.TIMELOW	:= T#500MS;
		Reset.LED				:= ResetLEDBlink.OUT;
END_CASE

HMI_Reset.LED := Reset.LED;
ResetLEDBlink(ENABLE := TRUE);

//Stop
CASE State OF
	E_State.Init..E_State.Enable:
		Stop.LED := FALSE;
	E_State.MoveToHome..E_State.CDoingWork:
		IF rtStop.Q THEN
			State := E_State.Stopping;
		END_IF

		Stop.LED := TRUE;
	E_State.Stopping:
		StopLEDBlink.TIMEHIGH	:= T#500MS;
		StopLEDBlink.TIMELOW	:= T#500MS;
		Stop.LED				:= StopLEDBlink.OUT;
	E_State.Stopped..E_State.Reseting:
		Stop.LED := FALSE;
END_CASE

HMI_Stop.LED := Stop.LED;
StopLEDBlink(ENABLE := TRUE);
END_METHOD

METHOD M_CloseGripper : BOOL
VAR_INPUT
END_VAR

VAR_INST
	tonDelay : TON;
END_VAR
tonDelay(IN := TRUE, PT := T#200MS);

Machine_D_Carrier_Gripper := TRUE;

IF tonDelay.Q THEN
	tonDelay(IN := FALSE);
	M_CloseGripper := TRUE;
END_IF
END_METHOD

METHOD M_HMI_Display
VAR_INPUT
END_VAR
(* Check if state has changed since the last cycle *)
IF lastState <> State THEN
	previousState := lastState; (* Update previous state *)
END_IF;

(* Update lastState for the next cycle *)
lastState := State;

//HMI Display strings
sPreviouseState	:= F_E_State_To_String(previousState);
sState			:= F_E_State_To_String(State);
sNextState		:= F_E_State_To_String(NextState);
END_METHOD

METHOD M_Init : BOOL
VAR_INPUT
END_VAR
VAR_INST
	InitStep : UDINT := 0;
END_VAR
CASE InitStep OF
	0://Create alarms
		//Estop buttons
		AlarmLocalEstopBtn.Arg1 := 'local';
		AlarmLocalEstopBtn.Create(EventEntry := TC_EVENTS.Safety.EstopBtn);
		AlarmAEstopBtn.Arg1 := 'A';
		AlarmAEstopBtn.Create(EventEntry := TC_EVENTS.Safety.EstopBtn);		
		AlarmBEstopBtn.Arg1 := 'B';
		AlarmBEstopBtn.Create(EventEntry := TC_EVENTS.Safety.EstopBtn);			
		AlarmCEstopBtn.Arg1 := 'C';
		AlarmCEstopBtn.Create(EventEntry := TC_EVENTS.Safety.EstopBtn);	
		AlarmDEstopBtn.Arg1 := 'D';
		AlarmDEstopBtn.Create(EventEntry := TC_EVENTS.Safety.EstopBtn);	
	
		//Light curtains
		AlarmALightCurtain.Arg1 := 'A';
		AlarmALightCurtain.Create(EventEntry := TC_EVENTS.Safety.LightCurtainTripped);	
		AlarmBLightCurtain.Arg1 := 'B';
		AlarmBLightCurtain.Create(EventEntry := TC_EVENTS.Safety.LightCurtainTripped);	
		AlarmCLightCurtain.Arg1 := 'C';
		AlarmCLightCurtain.Create(EventEntry := TC_EVENTS.Safety.LightCurtainTripped);

		//Axis
		AlarmXNotReady.Arg1 := 'X';
		AlarmXNotReady.Create(EventEntry := TC_EVENTS.DriveErrors.DriveHardwareNotReadyToOperate);					

		AlarmZNotReady.Arg1 := 'Z';
		AlarmZNotReady.Create(EventEntry := TC_EVENTS.DriveErrors.DriveHardwareNotReadyToOperate);

		AlarmXAxisError.Arg1 := 'X';
		AlarmXAxisError.Create(EventEntry := TC_EVENTS.DriveErrors.AxisInError);					

		AlarmZAxisError.Arg1 := 'Z';
		AlarmZAxisError.Create(EventEntry := TC_EVENTS.DriveErrors.AxisInError);
		
		AlarmAEstopTripped.Arg1 := 'A';
		AlarmAEstopTripped.Create(EventEntry := TC_EVENTS.Safety.MachineXEstopTripped);	
	
		AlarmBEstopTripped.Arg1 := 'B';
		AlarmBEstopTripped.Create(EventEntry := TC_EVENTS.Safety.MachineXEstopTripped);	
	
		AlarmCEstopTripped.Arg1 := 'C';
		AlarmCEstopTripped.Create(EventEntry := TC_EVENTS.Safety.MachineXEstopTripped);	
			
		AlarmDEstopTripped.Arg1 := 'D';
		AlarmDEstopTripped.Create(EventEntry := TC_EVENTS.Safety.MachineXEstopTripped);	
			
		InitStep := 20;
	20:
		M_Init := TRUE;
END_CASE
END_METHOD

METHOD M_OpenGripper : BOOL
VAR_INPUT
END_VAR
VAR_INST
	tonDelay : TON;
END_VAR
tonDelay(IN := TRUE, PT := T#200MS);
Machine_D_Carrier_Gripper := FALSE;

IF tonDelay.Q THEN
	tonDelay(IN := FALSE);
	M_OpenGripper := TRUE;
END_IF
END_METHOD

METHOD M_ProcessDelay : BOOL
VAR_INPUT
	pt : TIME;
END_VAR
VAR_INST
	tonDelay : TON;
END_VAR
tonDelay(IN := TRUE, PT := pt, Q =>, ET =>);

IF tonDelay.Q THEN
	M_ProcessDelay := TRUE;
	tonDelay(IN := FALSE, PT := pt, Q =>, ET =>);
END_IF
END_METHOD

METHOD M_ToTwinSAFE
VAR_INPUT
END_VAR
TwinSAFE_X_Axis_ActPos := TO_UDINT(X_Axis.NcToPlc.ActPos);

TwinSAFE_ResetAllEstopZones := Reset.Button OR HMI_Reset.Button;

TwinSAFEGroupRun := TRUE;
END_METHOD

END_FUNCTION_BLOCK

// ---- POUs/FB_Alarm.TcPOU
FUNCTION_BLOCK FB_Alarm
VAR_INPUT
	AlarmState : BOOL;
END_VAR
VAR_OUTPUT
END_VAR
VAR
	_hrAlarm		: HRESULT;
	_fbAlarm		: FB_TcAlarm;
	_EventEntry		: TcEventEntry;
	_Arg1, _Arg2	: STRING;
END_VAR


IF AlarmState THEN
	_fbAlarm.Raise(0);
ELSE
	_fbAlarm.Clear(0, 0);
END_IF

PROPERTY Arg1 : STRING
GET
Arg1 := _Arg1;
END_GET
SET
_Arg1 := Arg1;
END_SET
END_PROPERTY

PROPERTY Arg2 : STRING
GET
Arg2 := _Arg2;
END_GET
SET
_Arg2 := Arg2;
END_SET
END_PROPERTY

METHOD Create
VAR_INPUT
	EventEntry : TcEventEntry;
END_VAR
_EventEntry	:= EventEntry;
_hrAlarm	:= _fbAlarm.CreateEx(stEventEntry := EventEntry, bWithConfirmation := 0, ipSourceInfo := 0);

_fbAlarm.ipArguments.Clear();

IF _Arg1 <> '' THEN
	_fbAlarm.ipArguments.AddString(_Arg1);
END_IF

IF _Arg2 <> '' THEN
	_fbAlarm.ipArguments.AddString(_Arg2);
END_IF
END_METHOD

END_FUNCTION_BLOCK

// ---- POUs/F_E_State_To_String.TcPOU
//Convert E_Step to a string for display on the HMI
FUNCTION F_E_State_To_String : STRING
VAR_INPUT
	Step : E_State;
END_VAR
VAR
	StepString : STRING; // Adjust the size as needed
END_VAR


CASE Step OF
	E_State.Init:
		StepString := 'Init';
	E_State.Idel:
		StepString := 'Idle';
	E_State.Enable:
		StepString := 'Enable';
	E_State.MoveToHome:
		StepString := 'Move To Home';
	E_State.WaitForAToBeReady:
		StepString := 'Wait For A To Be Ready';
	E_State.MoveToAPickPos:
		StepString := 'Move To A Pick Position';
	E_State.PickFromA:
		StepString := 'Pick From A';
	E_State.MoveToBWaitPos:
		StepString := 'Move To B Wait Position';
	E_State.WaitForBToBeReady:
		StepString := 'Wait For B To Be Ready';
	E_State.MoveToBPlacePosition:
		StepString := 'Move To B Place Position';
	E_State.PlaceOnB:
		StepString := 'Place On B';
	E_State.MoveToBWorkPos:
		StepString := 'Move To B Work Position';
	E_State.BDoingWork:
		StepString := 'B Doing Work';
	E_State.MoveToBPickPos:
		StepString := 'Move To B Pick Position';
	E_State.PickPartFromB:
		StepString := 'Pick Part From B';
	E_State.MoveToCWaitPos:
		StepString := 'Move To C Wait Position';
	E_State.WaitForCToBeReady:
		StepString := 'Wait For C To Be Ready';
	E_State.MoveToCPlacePos:
		StepString := 'Move To C Place Position';
	E_State.PlaceOnC:
		StepString := 'Place On C';
	E_State.MoveToCWorkPos:
		StepString := 'Move To C Work Position';
	E_State.CDoingWork:
		StepString := 'C Doing Work';
	E_State.Stopping:
		StepString := 'Stopping';
	E_State.Stopped:
		StepString := 'Stopped';
	E_State.Error:
		StepString := 'Error';
	E_State.Reseting:
		StepString := 'Resetting';
ELSE
	StepString := 'Unknown';
END_CASE;

F_E_State_To_String := StepString;

END_FUNCTION

// ---- POUs/MAIN.TcPOU
PROGRAM MAIN
VAR
	Machine : FB_Machine;
END_VAR

PRG_LoadTwinSAFE();
Machine();

END_PROGRAM

// ---- POUs/PRG_LoadTwinSAFE.TcPOU
PROGRAM PRG_LoadTwinSAFE
VAR
	//On startup, check if the "correct" TwinSAFE program CRC is loaded.
	//System will restore it self back to "demo state" when powering up.
	
	LoaderAlarm				:FB_TcAlarm;
	
	Step					:(Init,WaitForOSToBoot,WaitForWcStateOk,CheckCRC,DownloadCode,Downloading,ActivateCode,Activating,Error,Done);
	tonWaitForOSToBoot		:TON:=(PT:=T#2M);
	ntCallTwinSAFELoader	:NT_StartProcess;
	ProjectCRC		AT%I*	:WORD;
	
	WcState			AT%I*	:BOOL;
	ManDownload				:BOOL;
	tonWait					:TON:=(PT:=T#10S);
	
END_VAR
VAR CONSTANT
	ExpectedProjectCRC		:WORD:=16#AAE7;
END_VAR


CASE Step OF
	Init:
		LoaderAlarm.CreateEx(stEventEntry := TC_EVENTS.Safety.TwinSAFELoaderError, bWithConfirmation := FALSE, ipSourceInfo := 0);
		Step := WaitForOSToBoot;

	WaitForOSToBoot:
		tonWaitForOSToBoot(IN := TRUE);

		IF tonWaitForOSToBoot.Q THEN
			Step := WaitForWcStateOk;
		END_IF

	WaitForWcStateOk:
		IF WcState = FALSE THEN
			Step := CheckCRC;
		END_IF

	CheckCRC:
		IF ProjectCRC = ExpectedProjectCRC THEN
			Step := Done;
		ELSE
			Step := DownloadCode;
		END_IF

	DownloadCode:
		ntCallTwinSAFELoader(NETID	:= '',
							PATHSTR := 'C:\TwinSAFE_Loader\TwinSAFE_Loader.exe',
							DIRNAME := 'C:\TwinSAFE_Loader\',
							COMNDLINE :=
							'--gw 172.16.17.50 --user Administrator --pass TwinSAFE --slave 1001 --proj C:\TwinSAFE_Loader\SafetyCode.bin',
							START := TRUE,
							TMOUT := T#15S);

		IF NOT ntCallTwinSAFELoader.BUSY THEN
			ntCallTwinSAFELoader(START := FALSE);

			IF NOT ntCallTwinSAFELoader.ERR THEN
				Step := Downloading;

			ELSE
				Step := Error;
				LoaderAlarm.ipArguments.Clear();
				LoaderAlarm.ipArguments.AddString('Downloading');
				LoaderAlarm.ipArguments.AddUDInt(ntCallTwinSAFELoader.ERRID);
			END_IF
		END_IF

	Downloading:
		tonWait(IN := TRUE);

		IF tonWait.Q THEN
			tonWait(IN := FALSE);
			Step := ActivateCode;
		END_IF

	ActivateCode:
		ntCallTwinSAFELoader(NETID	:= '',
							PATHSTR := 'C:\TwinSAFE_Loader\TwinSAFE_Loader.exe',
							DIRNAME := 'C:\TwinSAFE_Loader\',
							COMNDLINE :=
							'--gw 172.16.17.50 --user Administrator --pass TwinSAFE --slave 1001 --proj C:\TwinSAFE_Loader\SafetyCode.bin --crc 0xaae7',
							START := TRUE,
							TMOUT := T#15S);

		IF NOT ntCallTwinSAFELoader.BUSY THEN
			ntCallTwinSAFELoader(START := FALSE);

			IF NOT ntCallTwinSAFELoader.ERR THEN
				Step := Activating;
				ADSLOGSTR(msgCtrlMask := ADSLOG_MSGTYPE_LOG, msgFmtStr := 'TwinSAFE code has been activated', strArg := '');
			ELSE
				Step := Error;
				LoaderAlarm.ipArguments.Clear();
				LoaderAlarm.ipArguments.AddString('activating');
				LoaderAlarm.ipArguments.AddUDInt(ntCallTwinSAFELoader.ERRID);
			END_IF
		END_IF

	Activating:
		tonWait(IN := TRUE);

		IF tonWait.Q THEN
			tonWait(IN := FALSE);
			Step := Done;
		END_IF

	Error:
		IF ManDownload THEN
			ManDownload	:= FALSE;
			Step		:= DownloadCode;
		END_IF
	Done:
		IF ManDownload THEN
			ManDownload	:= FALSE;
			Step		:= DownloadCode;
		END_IF

END_CASE

END_PROGRAM
